// TIA Portal V16 export
// export: Created 2021-08-10T09:04:59.8372499Z, ExportSetting WithDefaults, WithReadOnly, DisplayName Totally Integrated Automation Portal, DisplayVersion V16, DisplayName TIA Portal Version Control Interface, DisplayVersion V16, DisplayName TIA Portal Openness, DisplayVersion V16, DisplayName TIA Portal Teamcenter Gateway, DisplayVersion V16, DisplayName SINAMICS Startdrive Advanced, DisplayVersion V16, DisplayName SINAMICS Startdrive G130, G150, S120, S150, SINAMICS MV, S210, DisplayVersion V16, DisplayName SINAMICS Startdrive G110M, G120, G120C, G120D, G120P, DisplayVersion V16, DisplayName STEP 7 Professional, DisplayVersion V16, DisplayName STEP 7 Safety, DisplayVersion V16, DisplayName WinCC Unified SCADA Engineering System, DisplayVersion V16
DATA_BLOCK "Valve Drain_DB"   // DB7
{ S7_Optimized_Access := 'TRUE' }
VERSION : 0.1
// stored: AutoNumber true, CodeModifiedDate 2020-02-26T12:49:16.2970167Z, CompileDate 2021-07-03T08:38:43.5846302Z, CreationDate 2020-02-26T12:48:12.3344036Z, DBAccessibleFromOPCUA true, DownloadWithoutReinit false, InstanceOfName Valve Drain, InstanceOfNumber 4, InstanceOfType FB, InterfaceModifiedDate 2020-02-26T12:48:59.514304Z, IsConsistent true, IsKnowHowProtected false, IsRetainMemResEnabled false, MemoryReserve 100, ModifiedDate 2020-02-26T12:49:16.2970167Z, ParameterModified 2020-02-26T07:16:51.9541274Z, StructureModified 2020-02-26T12:48:59.514304Z, UDAEnableTagReadback false
"Valve Drain"
   // VAR
   //    VlvDrn : "fbValve_Solenoid";
   // END_VAR
BEGIN
END_DATA_BLOCK
